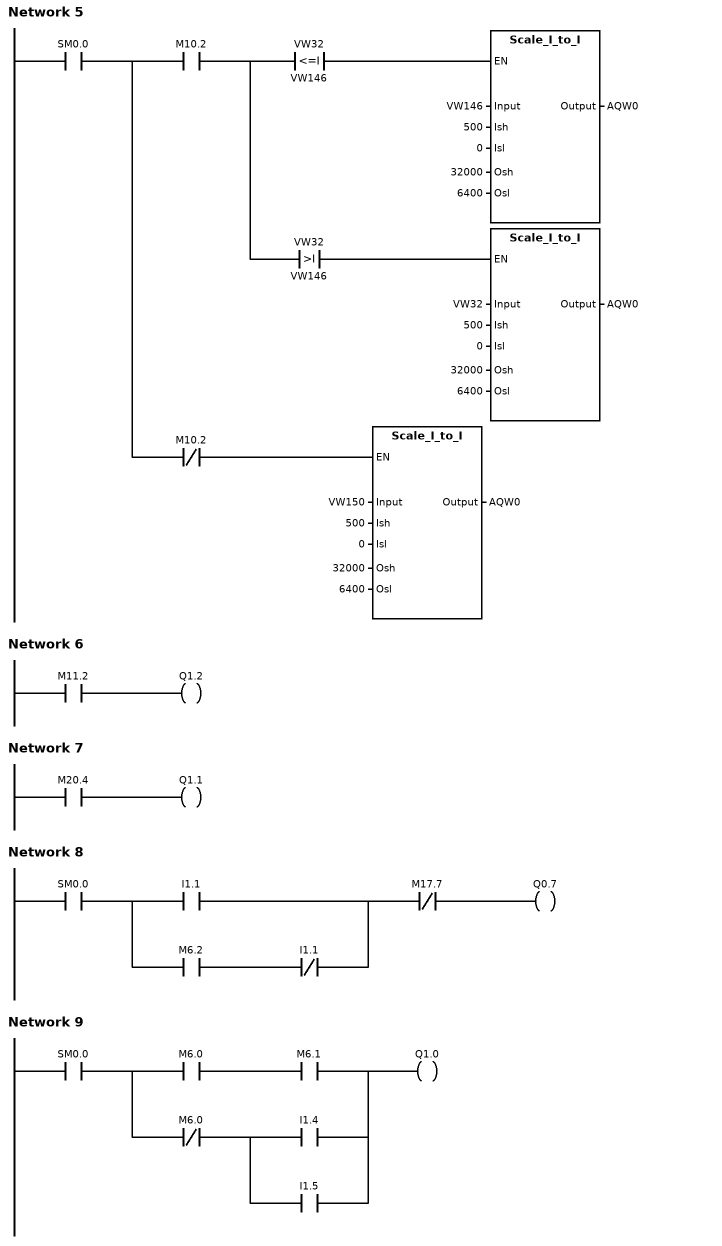
[picture p48: SBR24 networks 5-9]
Network 5
LD     SM0.0
LPS
A      M10.2
LPS
AW<=   VW32, VW146
CALL   Scale_I_to_I:SBR3, VW146, 500, 0, 32000, 6400, AQW0
LPP
AW>    VW32, VW146
CALL   Scale_I_to_I:SBR3, VW32, 500, 0, 32000, 6400, AQW0
LPP
AN     M10.2
CALL   Scale_I_to_I:SBR3, VW150, 500, 0, 32000, 6400, AQW0
Network 6
LD     M11.2
=      Q1.2
Network 7
LD     M20.4
=      Q1.1
Network 8
LD     SM0.0
LD     I1.1
LD     M6.2
AN     I1.1
OLD
ALD
AN     M17.7
=      Q0.7
Network 9
LD     SM0.0
LD     M6.0
A      M6.1
LDN    M6.0
LD     I1.4
O      I1.5
ALD
OLD
ALD
=      Q1.0
END_SUBROUTINE_BLOCK

SUBROUTINE_BLOCK SaveParameter:SBR26
TITLE=
BEGIN
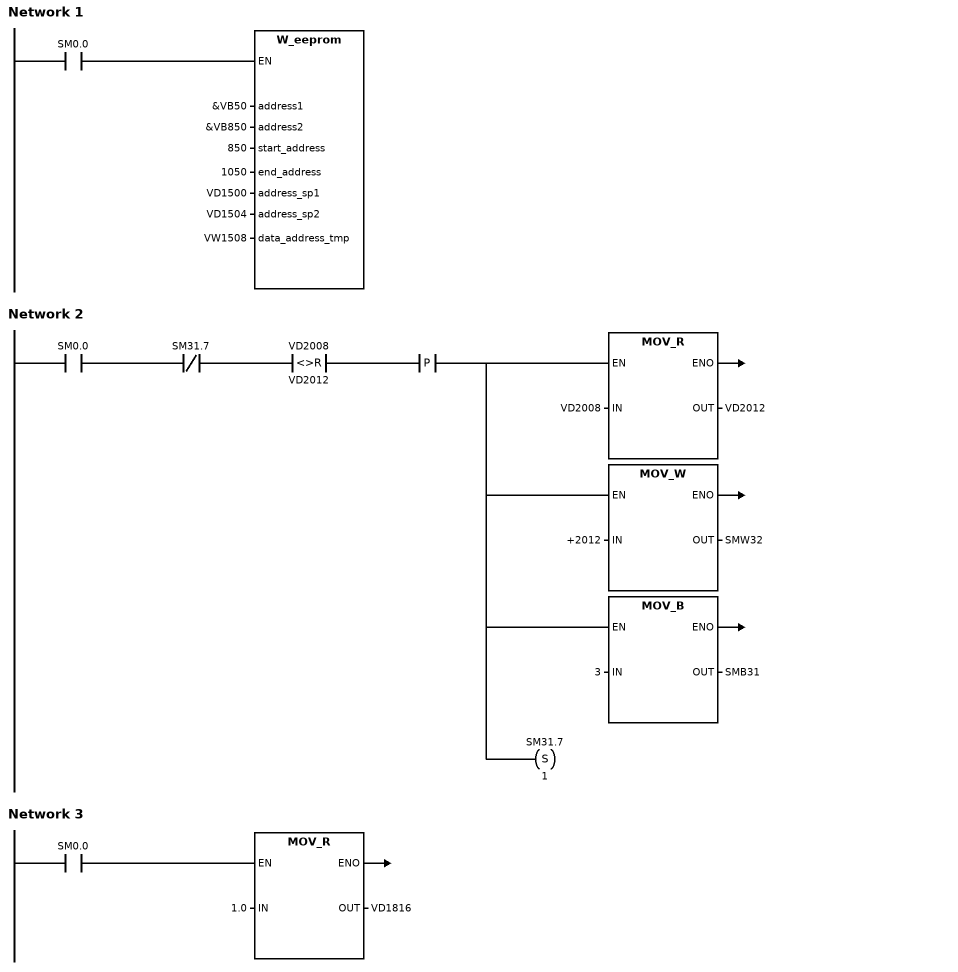
Network 1
LD     SM0.0
CALL   W_eeprom:SBR27, &VB50, &VB850, 850, 1050, VD1500, VD1504, VW1508
Network 2
LD     SM0.0
AN     SM31.7
AR<>   VD2008, VD2012
EU
MOVR   VD2008, VD2012
MOVW   +2012, SMW32
MOVB   3, SMB31
S      SM31.7, 1
Network 3
LD     SM0.0
MOVR   1.0, VD1816
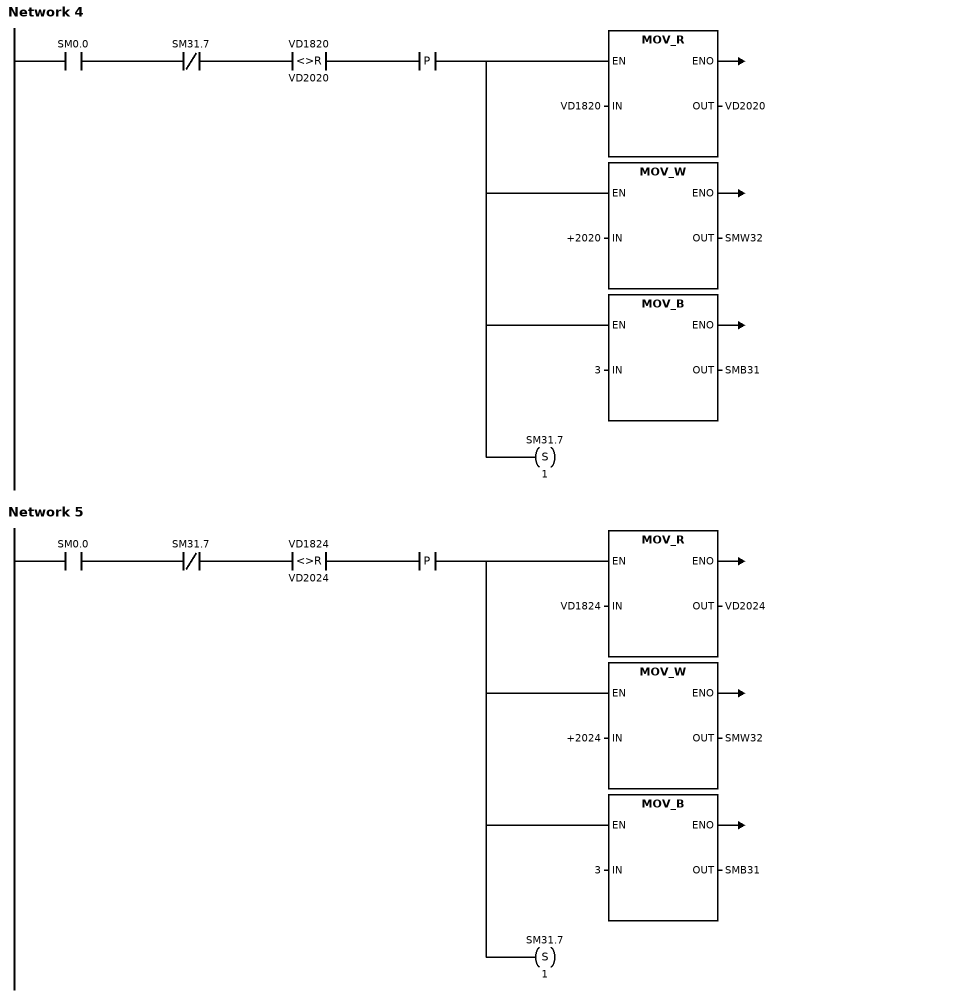
Network 4
LD     SM0.0
AN     SM31.7
AR<>   VD1820, VD2020
EU
MOVR   VD1820, VD2020
MOVW   +2020, SMW32
MOVB   3, SMB31
S      SM31.7, 1
Network 5
LD     SM0.0
AN     SM31.7
AR<>   VD1824, VD2024
EU
MOVR   VD1824, VD2024
MOVW   +2024, SMW32
MOVB   3, SMB31
S      SM31.7, 1
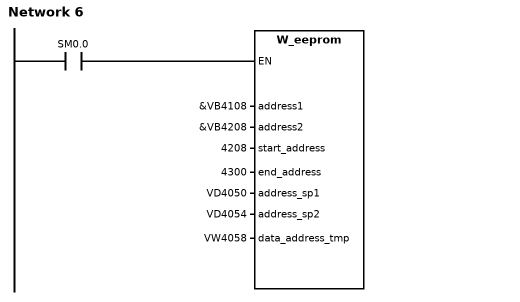
Network 6
LD     SM0.0
CALL   W_eeprom:SBR27, &VB4108, &VB4208, 4208, 4300, VD4050, VD4054, VW4058
END_SUBROUTINE_BLOCK

// SBR27: protected block, not included

SUBROUTINE_BLOCK KeyMain:SBR28
TITLE=
BEGIN
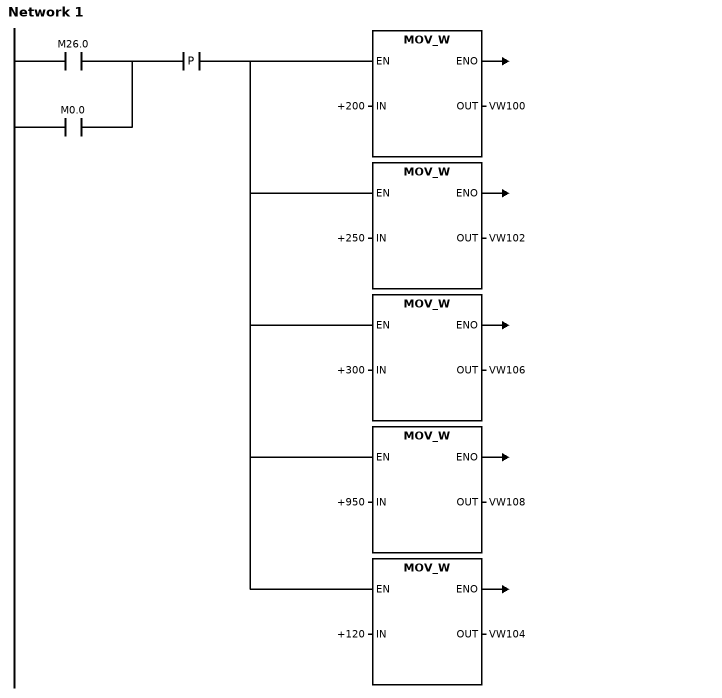
Network 1
LD     M26.0
O      M0.0
EU
MOVW   +200, VW100
MOVW   +250, VW102
MOVW   +300, VW106
MOVW   +950, VW108
MOVW   +120, VW104
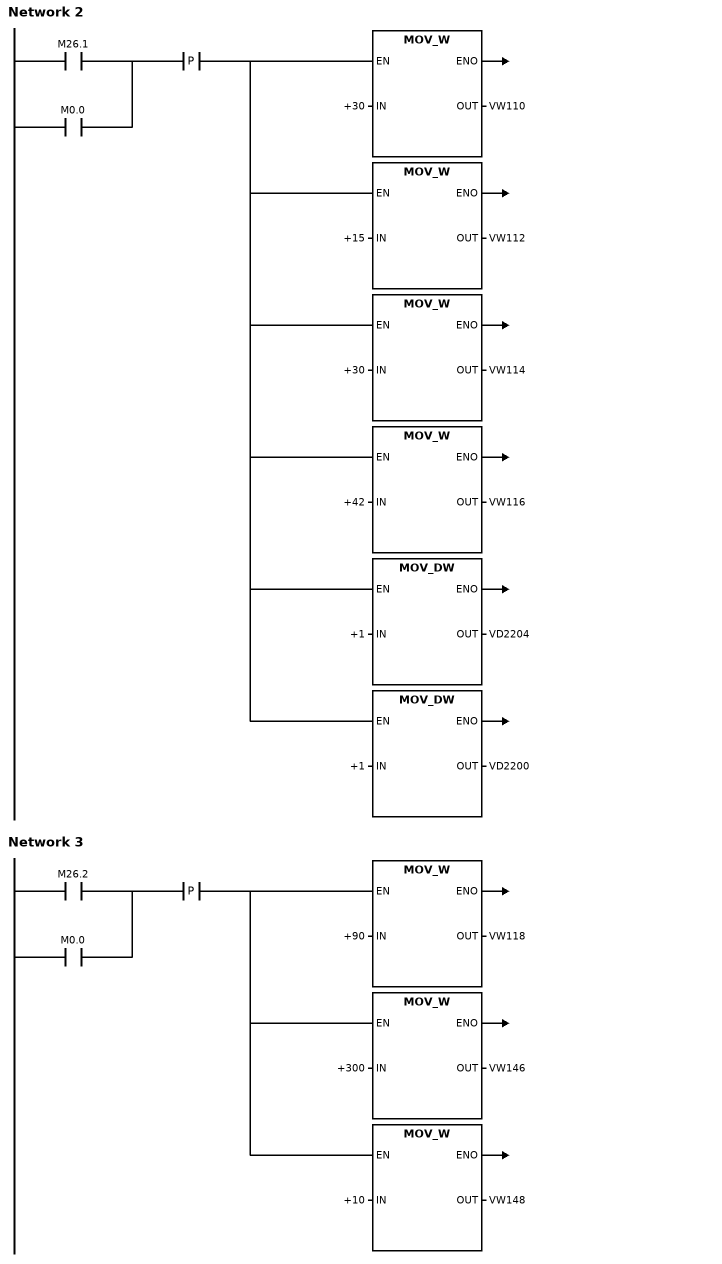
Network 2
LD     M26.1
O      M0.0
EU
MOVW   +30, VW110
MOVW   +15, VW112
MOVW   +30, VW114
MOVW   +42, VW116
MOVD   +1, VD2204
MOVD   +1, VD2200
Network 3
LD     M26.2
O      M0.0
EU
MOVW   +90, VW118
MOVW   +300, VW146
MOVW   +10, VW148
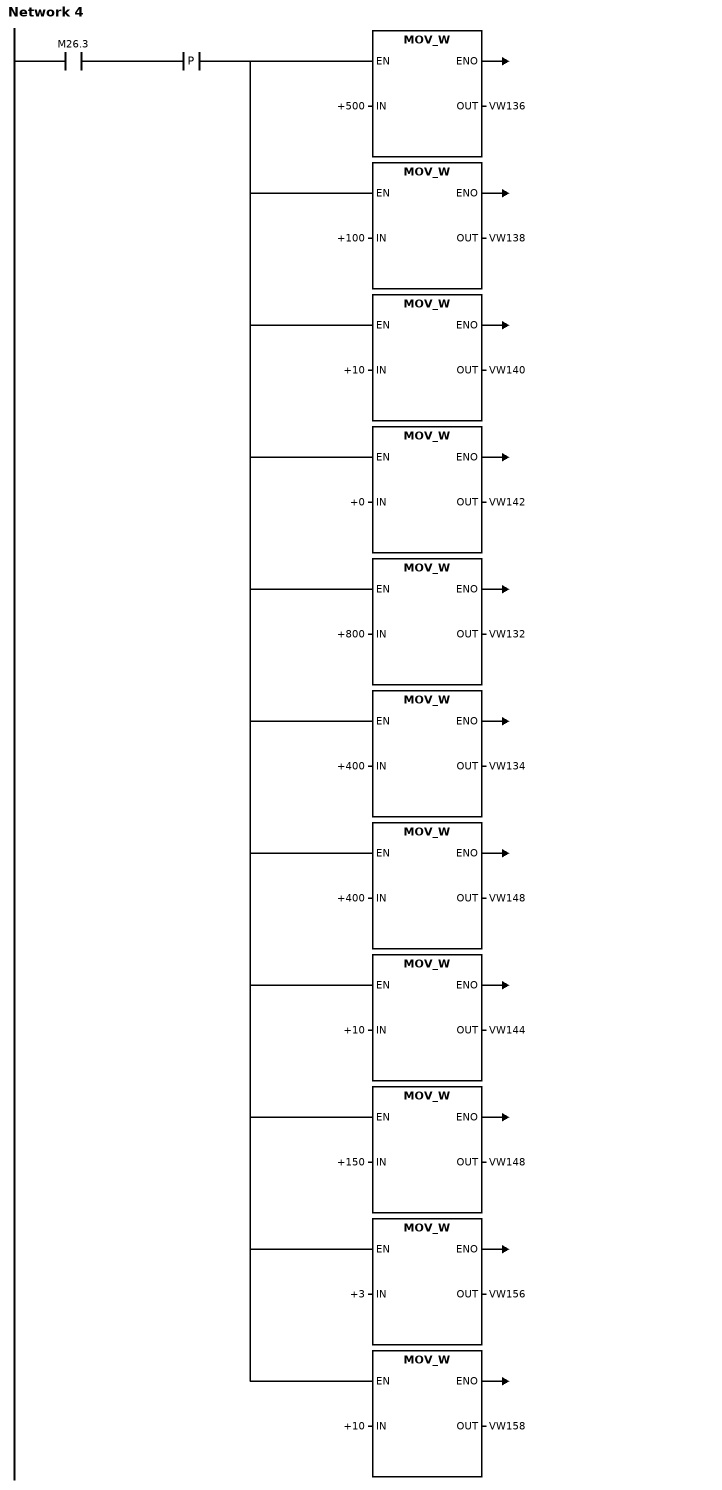
Network 4
LD     M26.3
EU
MOVW   +500, VW136
MOVW   +100, VW138
MOVW   +10, VW140
MOVW   +0, VW142
MOVW   +800, VW132
MOVW   +400, VW134
MOVW   +400, VW148
MOVW   +10, VW144
MOVW   +150, VW148
MOVW   +3, VW156
MOVW   +10, VW158
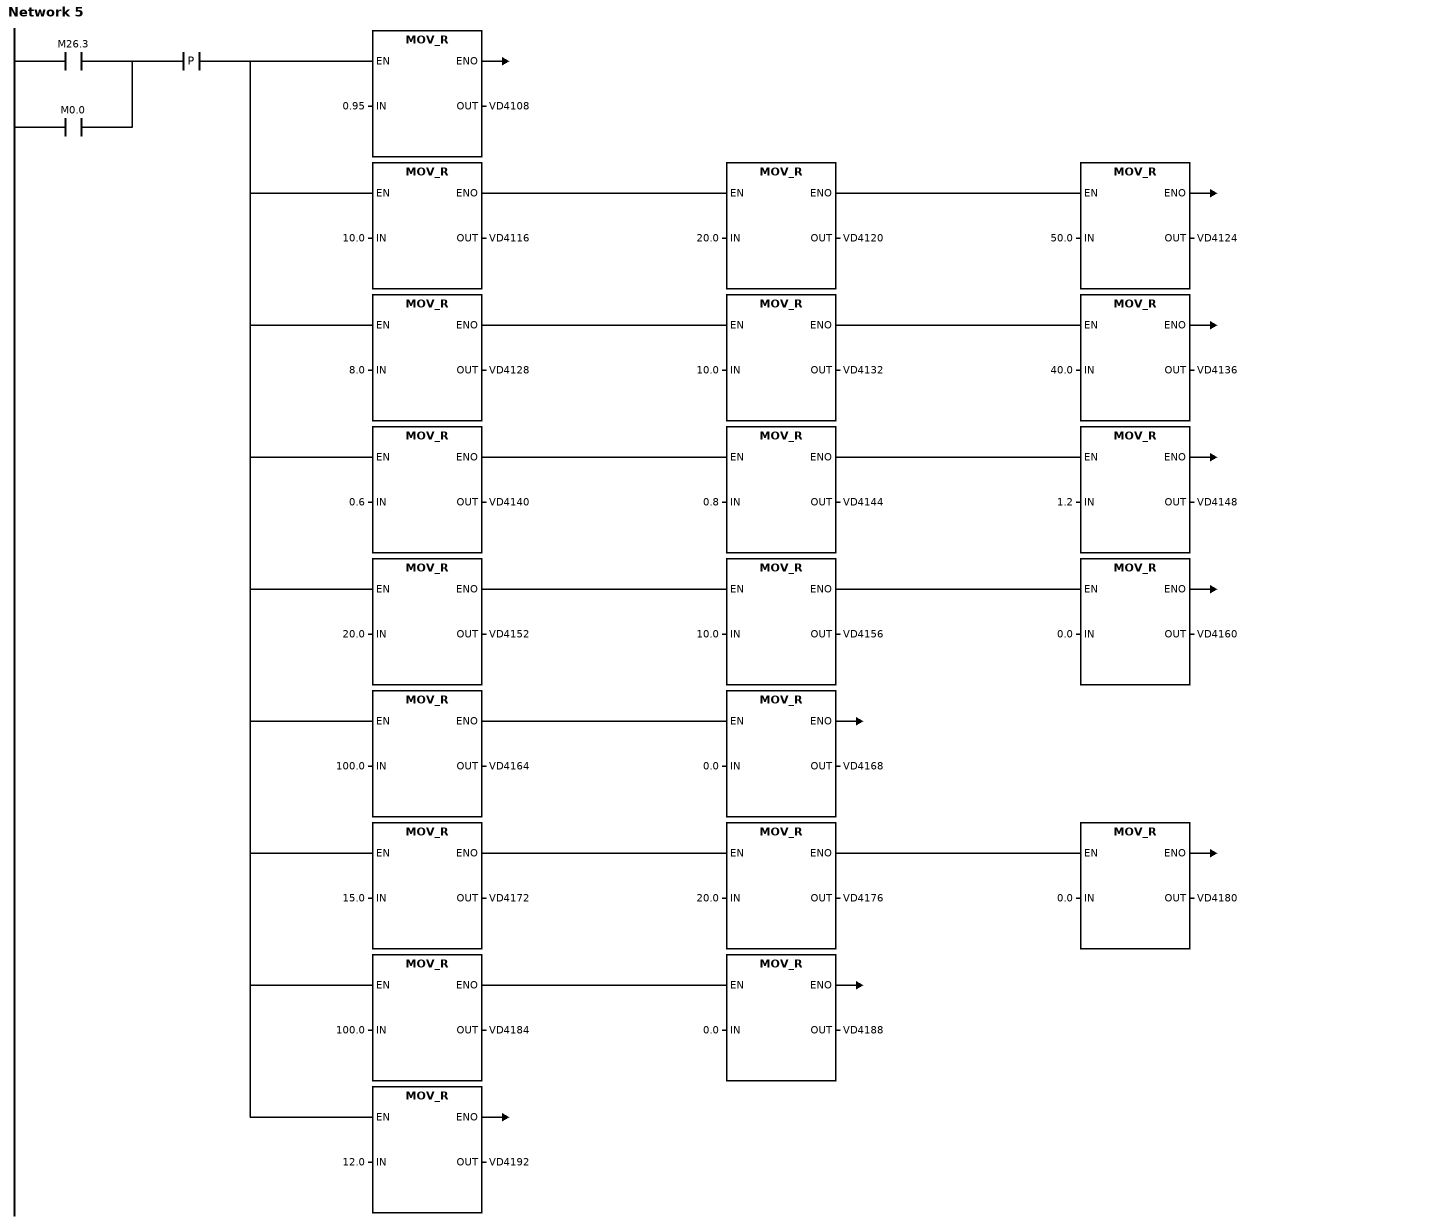
Network 5
LD     M26.3
O      M0.0
EU
LPS
MOVR   0.95, VD4108
MOVR   10.0, VD4116
AENO
MOVR   20.0, VD4120
AENO
MOVR   50.0, VD4124
LRD
MOVR   8.0, VD4128
AENO
MOVR   10.0, VD4132
AENO
MOVR   40.0, VD4136
LRD
MOVR   0.6, VD4140
AENO
MOVR   0.8, VD4144
AENO
MOVR   1.2, VD4148
LRD
MOVR   20.0, VD4152
AENO
MOVR   10.0, VD4156
AENO
MOVR   0.0, VD4160
LRD
MOVR   100.0, VD4164
AENO
MOVR   0.0, VD4168
LRD
MOVR   15.0, VD4172
AENO
MOVR   20.0, VD4176
AENO
MOVR   0.0, VD4180
LRD
MOVR   100.0, VD4184
AENO
MOVR   0.0, VD4188
LPP
MOVR   12.0, VD4192
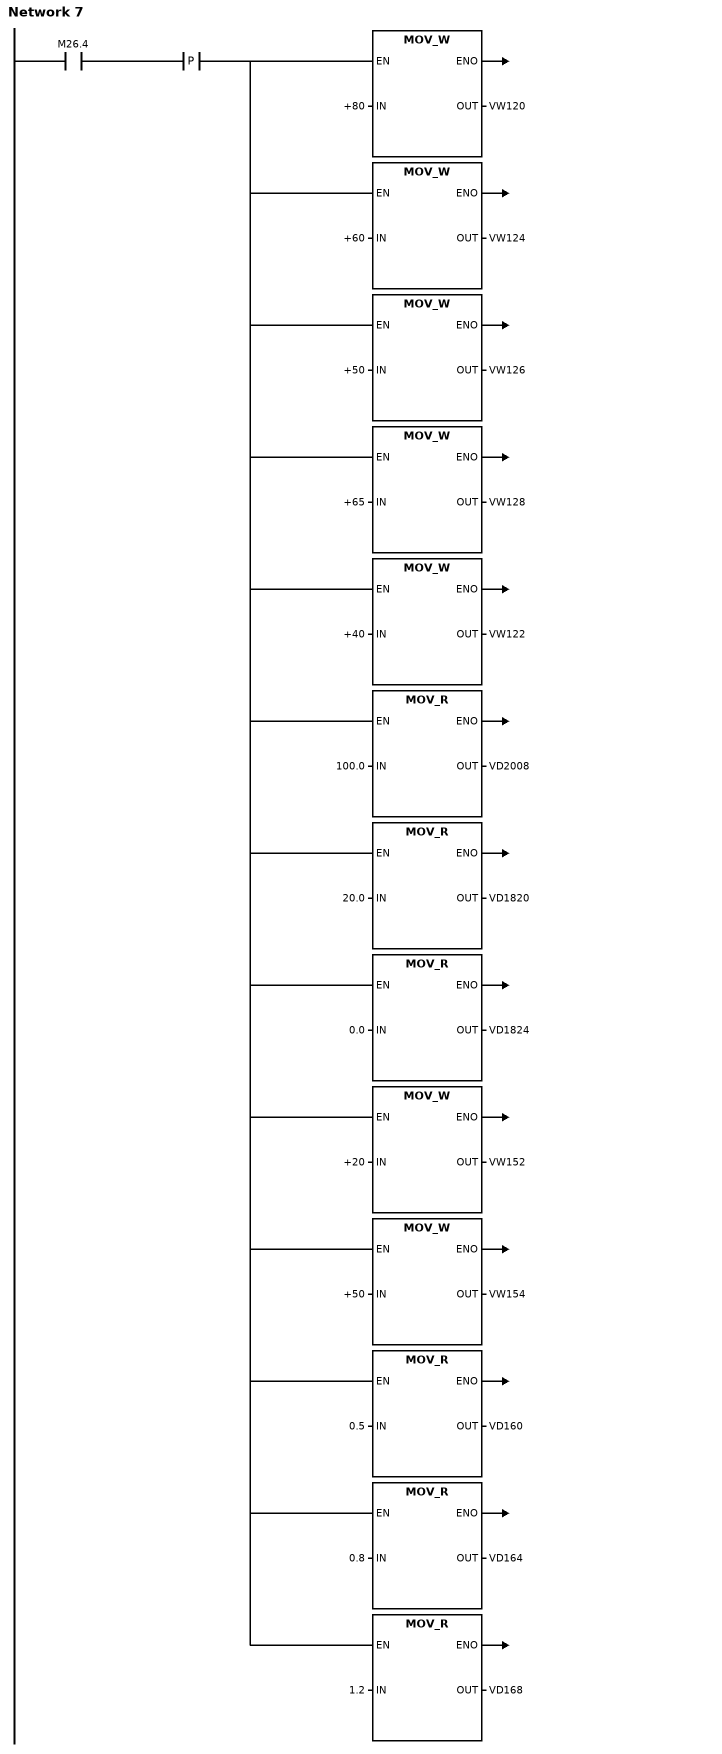
Network 7
LD     M26.4
EU
MOVW   +80, VW120
MOVW   +60, VW124
MOVW   +50, VW126
MOVW   +65, VW128
MOVW   +40, VW122
MOVR   100.0, VD2008
MOVR   20.0, VD1820
MOVR   0.0, VD1824
MOVW   +20, VW152
MOVW   +50, VW154
MOVR   0.5, VD160
MOVR   0.8, VD164
MOVR   1.2, VD168
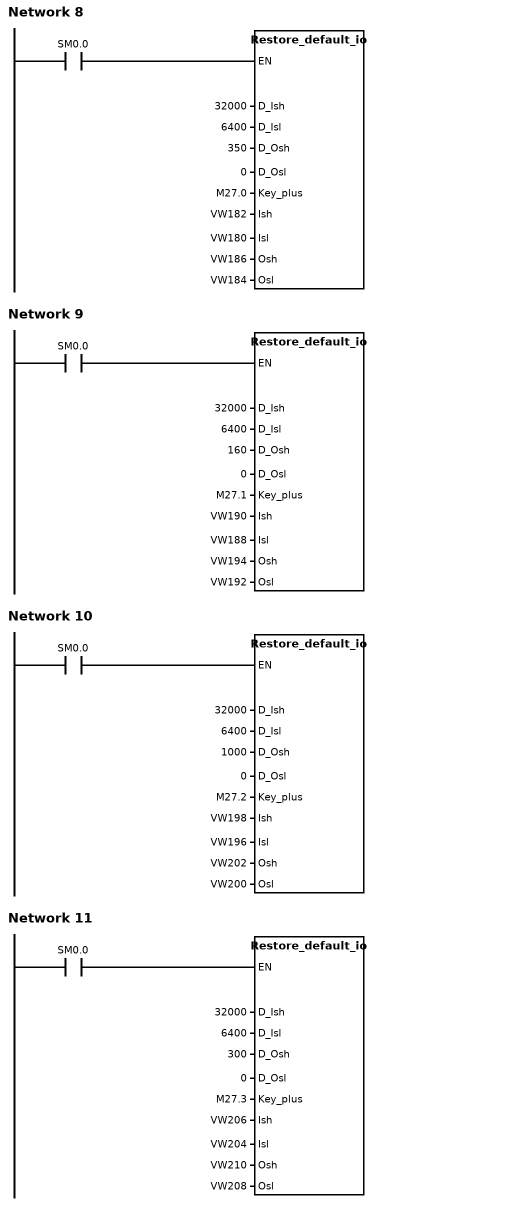
Network 8
LD     SM0.0
CALL   Restore_default_io:SBR29, 32000, 6400, 350, 0, M27.0, VW182, VW180, VW186, VW184
Network 9
LD     SM0.0
CALL   Restore_default_io:SBR29, 32000, 6400, 160, 0, M27.1, VW190, VW188, VW194, VW192
Network 10
LD     SM0.0
CALL   Restore_default_io:SBR29, 32000, 6400, 1000, 0, M27.2, VW198, VW196, VW202, VW200
Network 11
LD     SM0.0
CALL   Restore_default_io:SBR29, 32000, 6400, 300, 0, M27.3, VW206, VW204, VW210, VW208
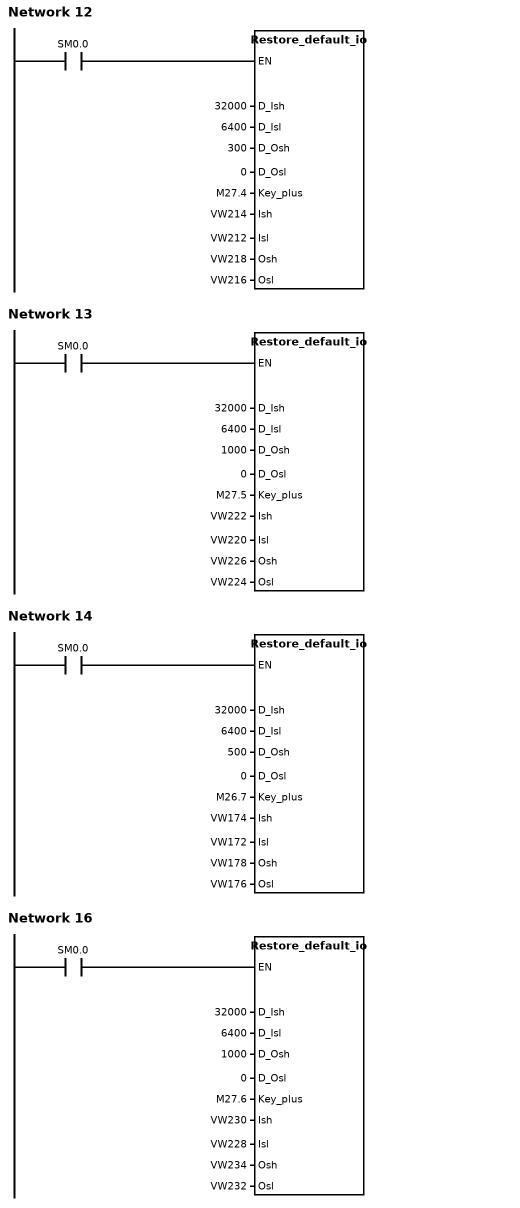
Network 12
LD     SM0.0
CALL   Restore_default_io:SBR29, 32000, 6400, 300, 0, M27.4, VW214, VW212, VW218, VW216
Network 13
LD     SM0.0
CALL   Restore_default_io:SBR29, 32000, 6400, 1000, 0, M27.5, VW222, VW220, VW226, VW224
Network 14
LD     SM0.0
CALL   Restore_default_io:SBR29, 32000, 6400, 500, 0, M26.7, VW174, VW172, VW178, VW176
Network 16
LD     SM0.0
CALL   Restore_default_io:SBR29, 32000, 6400, 1000, 0, M27.6, VW230, VW228, VW234, VW232
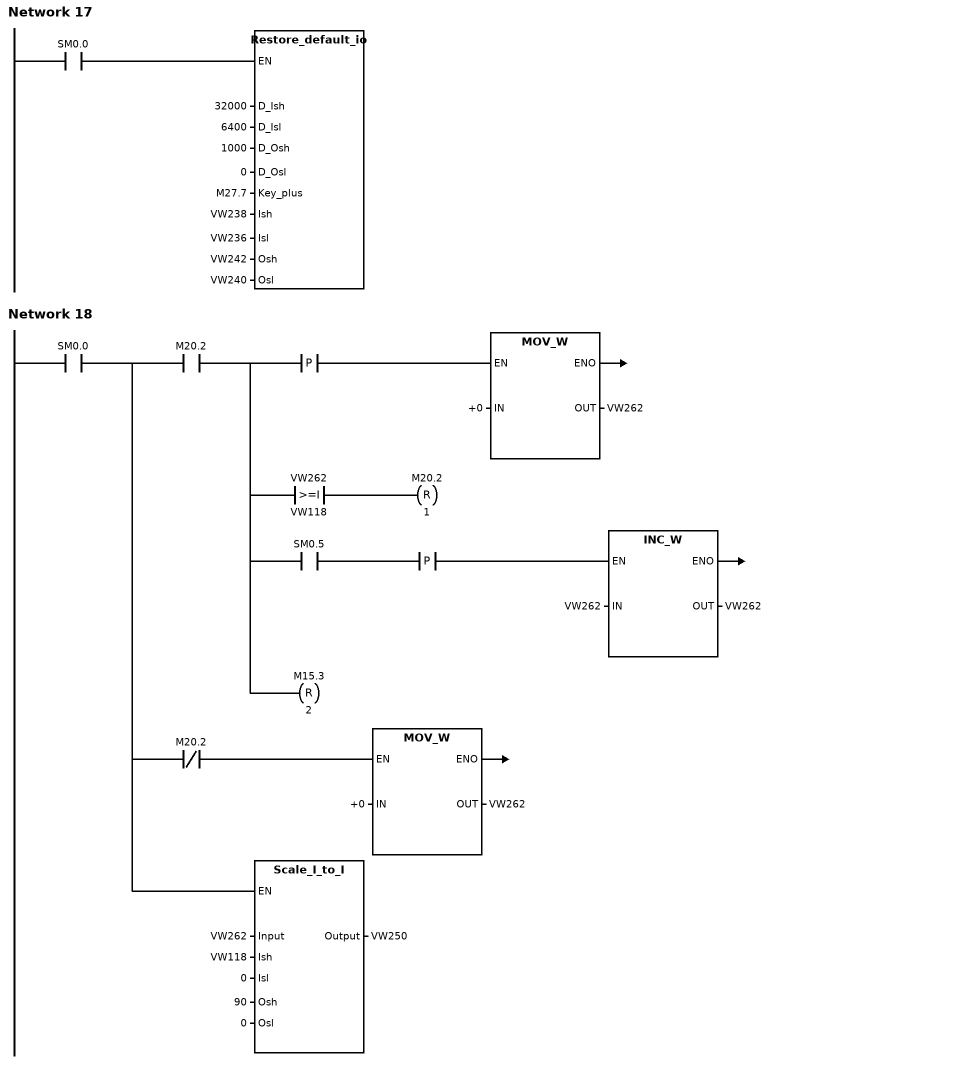
Network 17
LD     SM0.0
CALL   Restore_default_io:SBR29, 32000, 6400, 1000, 0, M27.7, VW238, VW236, VW242, VW240
Network 18
LD     SM0.0
LPS
A      M20.2
LPS
EU
MOVW   +0, VW262
LRD
AW>=   VW262, VW118
R      M20.2, 1
LRD
A      SM0.5
EU
INCW   VW262
LPP
R      M15.3, 2
LPP
LPS
AN     M20.2
MOVW   +0, VW262
LPP
CALL   Scale_I_to_I:SBR3, VW262, VW118, 0, 90, 0, VW250
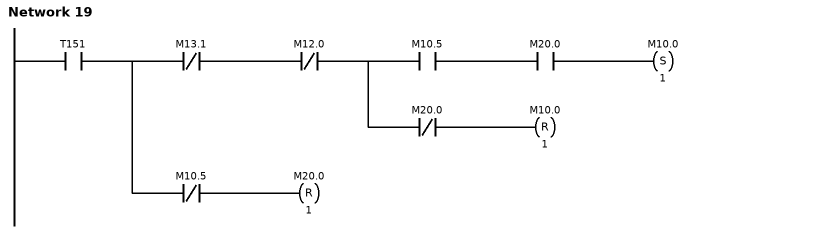
Network 19
LD     T151
LPS
AN     M13.1
AN     M12.0
LPS
A      M10.5
A      M20.0
S      M10.0, 1
LPP
AN     M20.0
R      M10.0, 1
LPP
AN     M10.5
R      M20.0, 1
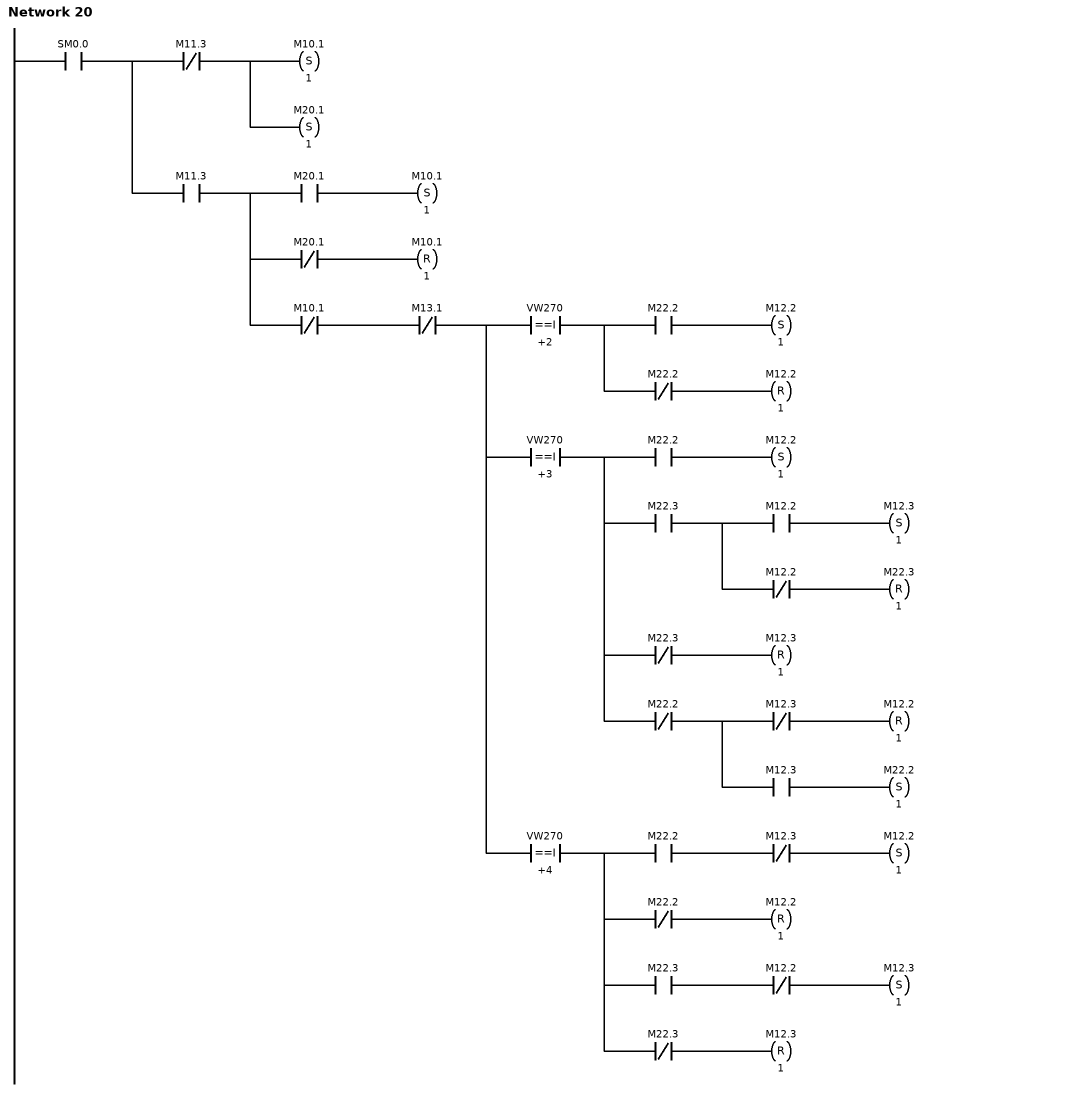
Network 20
LD     SM0.0
LPS
AN     M11.3
S      M10.1, 1
S      M20.1, 1
LPP
A      M11.3
LPS
A      M20.1
S      M10.1, 1
LRD
AN     M20.1
R      M10.1, 1
LPP
AN     M10.1
AN     M13.1
LPS
AW=    VW270, +2
LPS
A      M22.2
S      M12.2, 1
LPP
AN     M22.2
R      M12.2, 1
LRD
AW=    VW270, +3
LPS
A      M22.2
S      M12.2, 1
LRD
A      M22.3
LPS
A      M12.2
S      M12.3, 1
LPP
AN     M12.2
R      M22.3, 1
LRD
AN     M22.3
R      M12.3, 1
LPP
AN     M22.2
LPS
AN     M12.3
R      M12.2, 1
LPP
A      M12.3
S      M22.2, 1
LPP
AW=    VW270, +4
LPS
A      M22.2
AN     M12.3
S      M12.2, 1
LRD
AN     M22.2
R      M12.2, 1
LRD
A      M22.3
AN     M12.2
S      M12.3, 1
LPP
AN     M22.3
R      M12.3, 1
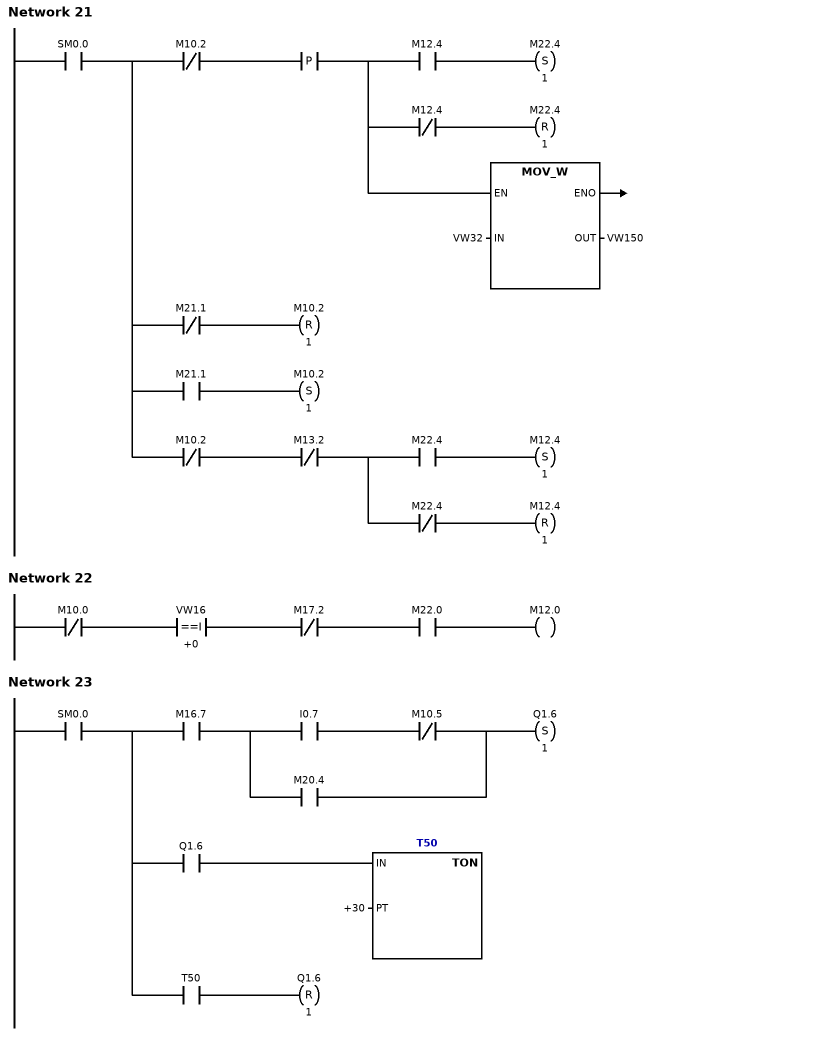
Network 21
LD     SM0.0
LPS
AN     M10.2
EU
LPS
A      M12.4
S      M22.4, 1
LRD
AN     M12.4
R      M22.4, 1
LPP
MOVW   VW32, VW150
LRD
LPS
AN     M21.1
R      M10.2, 1
LPP
A      M21.1
S      M10.2, 1
LPP
AN     M10.2
AN     M13.2
LPS
A      M22.4
S      M12.4, 1
LPP
AN     M22.4
R      M12.4, 1
Network 22
LDN    M10.0
AW=    VW16, +0
AN     M17.2
A      M22.0
=      M12.0
Network 23
LD     SM0.0
LPS
A      M16.7
LD     I0.7
AN     M10.5
O      M20.4
ALD
S      Q1.6, 1
LPP
LPS
A      Q1.6
TON    T50, +30
LPP
A      T50
R      Q1.6, 1
END_SUBROUTINE_BLOCK

// SBR29: protected block, not included

SUBROUTINE_BLOCK HcsCON:SBR32
TITLE=
BEGIN
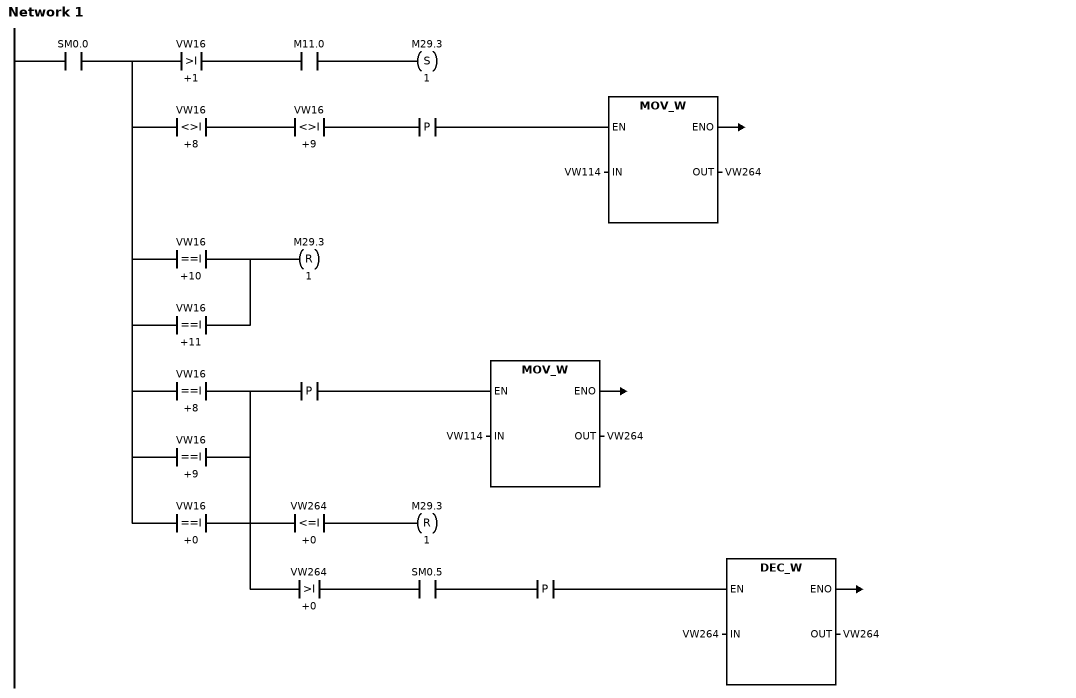
Network 1
LD     SM0.0
LPS
AW>    VW16, +1
A      M11.0
S      M29.3, 1
LRD
AW<>   VW16, +8
AW<>   VW16, +9
EU
MOVW   VW114, VW264
LRD
LDW=   VW16, +10
OW=    VW16, +11
ALD
R      M29.3, 1
LPP
LDW=   VW16, +8
OW=    VW16, +9
OW=    VW16, +0
ALD
LPS
EU
MOVW   VW114, VW264
LRD
AW<=   VW264, +0
R      M29.3, 1
LPP
AW>    VW264, +0
A      SM0.5
EU
DECW   VW264
END_SUBROUTINE_BLOCK

// SBR33: protected block, not included

// INT1: protected block, not included

// (further data pages could not be read)
